// TIA Portal V20 export
TYPE "LER_typeCmStatus"
// stored: Access Published
   STRUCT
      axisControl { ExternalWritable := 'False'} : Array[0..19] of "LBC_typeAxisControlNodeMonitoring";
      axis64Pos { ExternalWritable := 'False'} : Array[0..19] of "LBC_typeAxis64PosControlNodeMonitoring";
      twoWayAct { ExternalWritable := 'False'} : Array[0..19] of "LBC_typeTwoWayActuatorControlNodeMonitoring";
      digitalSignal { ExternalWritable := 'False'} : Array[0..19] of "LBC_typeDigitalSignalControlNodeMonitoring";
   END_STRUCT;
END_TYPE
